# EPICS StreamDevice protocol: ioc/protocol/SGA.proto
Terminator = CR LF;

getInfo{
#	@init {
#		out "*CLS";
#		out "*RST";
#	}
	out "IDN?"; in "%s";
}

setRemote{
	@init {
		out "*CLS";
		out "*RST";
	}
	out "SYST:LOCAL 0";
}

getRemote{
#	@init {
#		out "*CLS";
#		out "*RST";
#	}
	out "SYST:LOCAL?"; in "%i";
}

setCurrent{
#	@init {
#		out "*CLS";
#		out "*RST";
#	}
	out "SOUR:CURR 188.0";
}

getCurrent{
#	@init {
#		out "*CLS";
#		out "*RST";
#	}
	out "SOURCE:CURRENT?"; in "%f";
}

setVoltageZero{
#	@init {
#		out "*CLS";
#		out "*RST";
#	}
	out "SOUR:VOLT 0.0";
}

getVoltage{
#	@init {
#		out "*CLS";
#		out "*RST";
#	}
	out "SOURCE:VOLTAGE?"; in "%f";
}

setProtVoltage{
#	@init {
#		out "*CLS";
#		out "*RST";
#	}
	out "SOUR:VOLT:PROT 88.0";
}

getProtVoltage{
#	@init {
#		out "*CLS";
#		out "*RST";
#	}
	out "SOUR:VOLT:PROT?"; in "%f";
}

getOutCurrent{
#	@init {
#		out "*CLS";
#		out "*RST";
#	}
	out "MEASURE:CURRENT?"; in "%f";
}

getOutVoltage{
#	@init {
#		out "*CLS";
#		out "*RST";
#	}
	out "MEASURE:VOLTAGE?"; in "%f";
}

getOutPower{
#	@init {
#		out "*CLS";
#		out "*RST";
#	}
	out "MEASURE:POWER?"; in "%f";
}

getStatus{
#	@init {
#		out "*CLS";
#		out "*RST";
#	}
	out "OUTP:STAT?"; in "%i";
}

setOutOff{
#	@init {
#		out "*CLS";
#		out "*RST";
#	}
	out "OUTP:STAT OFF";
}

setOutOn{
#	@init {
#		out "*CLS";
#		out "*RST";
#	}
	out "OUTP:STAT ON";
}
